% RSLogix 500 project Q8.RSS, saved by version 8.30.00.16 %
PROJECT "Q8"    % processor: Bul.1763 MicroLogix 1100 Series B %

PROGRAM FILES
  LAD 2   7 rungs

DATA FILES
  O0 OUTPUT  4 elements
  I1 INPUT  6 elements
  S2 STATUS  66 elements
  B3 BINARY  1 elements
  T4 TIMER  1 elements
  C5 COUNTER  1 elements
  R6 CONTROL  1 elements
  N7 INTEGER  1 elements
  F8 FLOAT  1 elements

LADDER 2
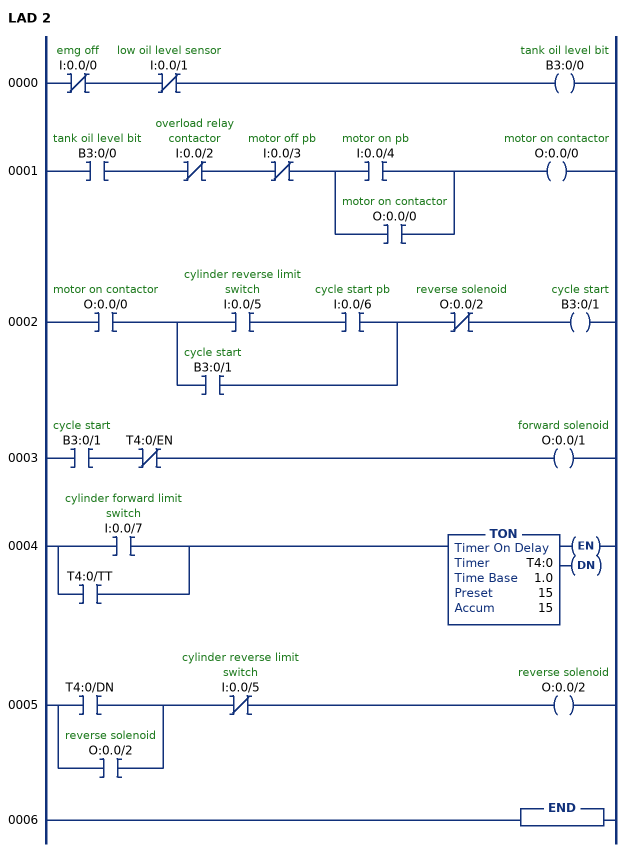
% Rung: 0 %
SOR XIO I:0.0/0 XIO I:0.0/1 OTE B3:0/0 EOR
%   I:0.0/0  "emg off" %
%   I:0.0/1  "low oil level sensor" %
%   B3:0/0  "tank oil level bit" %
% Rung: 1 %
SOR XIC B3:0/0 XIO I:0.0/2 XIO I:0.0/3 BST XIC I:0.0/4 NXB XIC O:0.0/0 BND OTE O:0.0/0 EOR
%   B3:0/0  "tank oil level bit" %
%   I:0.0/2  "overload relay contactor" %
%   I:0.0/3  "motor off pb" %
%   I:0.0/4  "motor on pb" %
%   O:0.0/0  "motor on contactor" %
% Rung: 2 %
SOR XIC O:0.0/0 BST XIC I:0.0/5 XIC I:0.0/6 NXB XIC B3:0/1 BND XIO O:0.0/2 OTE B3:0/1 EOR
%   O:0.0/0  "motor on contactor" %
%   I:0.0/5  "cylinder reverse limit switch" %
%   I:0.0/6  "cycle start pb" %
%   B3:0/1  "cycle start" %
%   O:0.0/2  "reverse solenoid" %
% Rung: 3 %
SOR XIC B3:0/1 XIO T4:0/EN OTE O:0.0/1 EOR
%   B3:0/1  "cycle start" %
%   O:0.0/1  "forward solenoid" %
% Rung: 4 %
SOR BST XIC I:0.0/7 NXB XIC T4:0/TT BND TON T4:0 1.0 15 15 EOR
%   I:0.0/7  "cylinder forward limit switch" %
% Rung: 5 %
SOR BST XIC T4:0/DN NXB XIC O:0.0/2 BND XIO I:0.0/5 OTE O:0.0/2 EOR
%   O:0.0/2  "reverse solenoid" %
%   I:0.0/5  "cylinder reverse limit switch" %
% Rung: 6 %
SOR END EOR

DATA TABLE (non-zero values as saved)
DATA B3
% B3:0 % 0X0003
DATA T4
% .PRE .ACC %
% T4:0 % 15 15
